1600, txt_DbVar_C1_NvParametersC1_MaxPvgRotTurretCtClkwseRadioPost_0 := 1601, txt_DbVarArrDescr_C1_NvParametersC1_RotTurretCtClkwiseRampRatioTuret := 1602, txt_DbVar_C1_NvParametersC1_RotTurretCtClkwiseRampRatioTuret_0 := 1603, txt_DbVar_C1_NvParametersC1_RotTurretCtClkwiseRampRatioTuret_1 := 1604, txt_DbVarArrDescr_C1_NvParametersC1_RotTurretCtClkwiseRampRatioNacel := 1605, txt_DbVar_C1_NvParametersC1_RotTurretCtClkwiseRampRatioNacel_0 := 1606, txt_DbVar_C1_NvParametersC1_RotTurretCtClkwiseRampRatioNacel_1 := 1607, txt_DbVarArrDescr_C1_NvParametersC1_RotTurretCtClkwiseRampRatioRadio := 1608, txt_DbVar_C1_NvParametersC1_RotTurretCtClkwiseRampRatioRadio_0 := 1609, txt_DbVar_C1_NvParametersC1_RotTurretCtClkwiseRampRatioRadio_1 := 1610, txt_DbVar_C1_NvParametersC1_MinPvgUpAxleOscillant_0 := 1611, txt_DbVar_C1_NvParametersC1_MaxPvgUpAxleOscillant_0 := 1612, txt_DbVarArrDescr_C1_NvParametersC1_PvgUpAxleOscillantRampRatio := 1613, txt_DbVar_C1_NvParametersC1_PvgUpAxleOscillantRampRatio_0 := 1614, txt_DbVar_C1_NvParametersC1_PvgUpAxleOscillantRampRatio_1 := 1615, txt_DbVar_C1_NvParametersC1_MinPvgDownAxleOscillant_0 := 1616, txt_DbVar_C1_NvParametersC1_MaxPvgDownAxleOscillant_0 := 1617, txt_DbVarArrDescr_C1_NvParametersC1_PvgDownAxleOscillantRampRatio := 1618, txt_DbVar_C1_NvParametersC1_PvgDownAxleOscillantRampRatio_0 := 1619, txt_DbVar_C1_NvParametersC1_PvgDownAxleOscillantRampRatio_1 := 1620, txt_DbVar_C1_NvParametersC1_MinPvgUpAxleFixe_0 := 1621, txt_DbVar_C1_NvParametersC1_MaxPvgUpAxleFixe_0 := 1622, txt_DbVarArrDescr_C1_NvParametersC1_PvgUpAxleFixeRampRatio := 1623, txt_DbVar_C1_NvParametersC1_PvgUpAxleFixeRampRatio_0 := 1624, txt_DbVar_C1_NvParametersC1_PvgUpAxleFixeRampRatio_1 := 1625, txt_DbVar_C1_NvParametersC1_MinPvgDownAxleFixe_0 := 1626, txt_DbVar_C1_NvParametersC1_MaxPvgDownAxleFixe_0 := 1627, txt_DbVarArrDescr_C1_NvParametersC1_PvgDownAxleFixeRampRatio := 1628, txt_DbVar_C1_NvParametersC1_PvgDownAxleFixeRampRatio_0 := 1629, txt_DbVar_C1_NvParametersC1_PvgDownAxleFixeRampRatio_1 := 1630, txt_DbVar_C1_NvParametersC1_MinPvgRotFrameCtClkwise_0 := 1631, txt_DbVar_C1_NvParametersC1_MaxPvgRotFrameCtClkwise_0 := 1632, txt_DbVarArrDescr_C1_NvParametersC1_RotFrameCtClkwiseRampRatio := 1633, txt_DbVar_C1_NvParametersC1_RotFrameCtClkwiseRampRatio_0 := 1634, txt_DbVar_C1_NvParametersC1_RotFrameCtClkwiseRampRatio_1 := 1635, txt_DbVar_C1_NvParametersC1_MinPvgRotFrameClkwise_0 := 1636, txt_DbVar_C1_NvParametersC1_MaxPvgRotFrameClkwise_0 := 1637, txt_DbVarArrDescr_C1_NvParametersC1_RotFrameClkwiseRampRatio := 1638, txt_DbVar_C1_NvParametersC1_RotFrameClkwiseRampRatio_0 := 1639, txt_DbVar_C1_NvParametersC1_RotFrameClkwiseRampRatio_1 := 1640, txt_DbVar_C1_NvParametersC1_AntiDemarrageTime_0 := 1641, txt_DbVar_C1_NvParametersC1_TresholdRmpMotorAntidemarrage_0 := 1642, txt_DbVar_C1_NvParametersC1_SlowSpeedUpDeltaArmTelescOut_0 := 1643, txt_DbVar_C1_NvParametersC1_SlowSpeedDownDeltaArmTelescOut_0 := 1644, txt_DbVar_C1_NvParametersC1_SlowSpeedUpArrowArmTelescOut_0 := 1645, txt_DbVar_C1_NvParametersC1_SlowSpeedDownArrowArmTelescOut_0 := 1646, txt_DbVar_C1_NvParametersC1_RotTurretClockSlowSpeedRedAlo_0 := 1647, txt_DbVar_C1_NvParametersC1_RotTurretCtClockSlowSpeedRedAlo_0 := 1648, txt_DbVar_C1_NvParametersC1_ArrowArmDownSlowSpeedRedAlo_0 := 1649, txt_DbVar_C1_NvParametersC1_SlowSpeedRotTurretCtClokTelecOut_0 := 1650, txt_DbVar_C1_NvParametersC1_SlowSpeedRotTurretClokTelecOut_0 := 1651, txt_DbVar_C1_NvParametersC1_MinPvgUpMastMeasure_0 := 1652, txt_DbVar_C1_NvParametersC1_MaxPvgUpMastMeasure_0 := 1653, txt_DbVarArrDescr_C1_NvParametersC1_UpMastMeasureRampRatio := 1654, txt_DbVar_C1_NvParametersC1_UpMastMeasureRampRatio_0 := 1655, txt_DbVar_C1_NvParametersC1_UpMastMeasureRampRatio_1 := 1656, txt_DbVar_C1_NvParametersC1_MinPvgDownMastMeasure_0 := 1657, txt_DbVar_C1_NvParametersC1_MaxPvgDownMastMeasure_0 := 1658, txt_DbVarArrDescr_C1_NvParametersC1_DownMastMeasureRampRatio := 1659, txt_DbVar_C1_NvParametersC1_DownMastMeasureRampRatio_0 := 1660, txt_DbVar_C1_NvParametersC1_DownMastMeasureRampRatio_1 := 1661, txt_DbVar_C1_NvParametersC1_OutCharPosTransmission1Pressure_0 := 1662, txt_DbVar_C1_NvParametersC1_OutCharNeuTransmission1Pressure_0 := 1663, txt_DbVar_C1_NvParametersC1_OutCharNegTransmission1Pressure_0 := 1664, txt_DbVar_C1_NvParametersC1_InCharPosTransmission1Pressure_0 := 1665, txt_DbVar_C1_NvParametersC1_InCharNeuTransmission1Pressure_0 := 1666, txt_DbVar_C1_NvParametersC1_INCharNegTransmission1Pressure_0 := 1667, txt_DbVar_C1_NvParametersC1_OutCharPosTransmission2Pressure_0 := 1668, txt_DbVar_C1_NvParametersC1_OutCharNeuTransmission2Pressure_0 := 1669, txt_DbVar_C1_NvParametersC1_OutCharNegTransmission2Pressure_0 := 1670, txt_DbVar_C1_NvParametersC1_InCharPosTransmission2Pressure_0 := 1671, txt_DbVar_C1_NvParametersC1_InCharNeuTransmission2Pressure_0 := 1672, txt_DbVar_C1_NvParametersC1_INCharNegTransmission2Pressure_0 := 1673, txt_DbVar_C1_NvParametersC1_OutCharPosBypassPressureSensor_0 := 1674, txt_DbVar_C1_NvParametersC1_OutCharNeuBypassPressureSensor_0 := 1675, txt_DbVar_C1_NvParametersC1_OutCharNegBypassPressureSensor_0 := 1676, txt_DbVar_C1_NvParametersC1_InCharPosBypassPressureSensor_0 := 1677, txt_DbVar_C1_NvParametersC1_InCharNeuBypassPressureSensor_0 := 1678, txt_DbVar_C1_NvParametersC1_InCharNegBypassPressureSensor_0 := 1679, txt_DbVar_C1_NvParametersC1_NvParametersC1_1_0 := 1680, txt_DbVar_C1_NvParametersC1_NvParametersC1_2_0 := 1681, txt_DbVar_C1_NvParametersC1_NvParametersC1_3_0 := 1682, txt_DbVar_C1_NvParametersC1_NvParametersC1_4_0 := 1683, txt_DbVar_C1_NvParametersC1_NvParametersC1_5_0 := 1684, txt_DbVar_C1_NvParametersC1_NvParametersC1_6_0 := 1685, txt_DbVar_C1_NvParametersC1_NvParametersC1_7_0 := 1686, txt_DbVar_C1_NvParametersC1_NvParametersC1_8_0 := 1687, txt_DbVar_C1_NvParametersC1_NvParametersC1_9_0 := 1688, txt_DbVar_C1_NvParametersC1_NvParametersC1_10_0 := 1689, txt_DbVar_C1_NvParametersC1_NvParametersC1_11_0 := 1690, txt_DbVar_C1_NvParametersC1_NvParametersC1_12_0 := 1691, txt_DbVar_C1_NvParametersC1_NvParametersC1_13_0 := 1692, txt_DbVar_C1_NvParametersC1_NvParametersC1_14_0 := 1693, txt_DbVar_C1_NvParametersC1_NvParametersC1_15_0 := 1694, txt_DbVar_C1_NvParametersC1_NvParametersC1_16_0 := 1695, txt_DbVar_C1_NvParametersC1_NvParametersC1_17_0 := 1696, txt_DbVar_C1_NvParametersC1_CurFor220VGeneratorOn_0 := 1697, txt_DbVar_C1_NvParametersC1_NbElementTransissionPressure_0 := 1698, txt_DbVar_C1_NvParametersC1_RampUpEvGenerator_0 := 1699, txt_DbVar_C1_NvParametersC1_RampDownEvGenerator_0 := 1700, txt_DbVar_C1_NvParametersC1_GasGaugeAlarm_0 := 1701, txt_DbVar_C1_NvParametersC1_CRC_SRDO1_0 := 1702, txt_DbVar_C1_NvParametersC1_CRC_SRDO2_0 := 1703, txt_DbVar_C1_NvParametersC1_CRC_SRDO3_0 := 1704, txt_DbVar_C1_NvParametersC1_CRC_SRDO4_0 := 1705, txt_DbVar_C1_NvParametersC1_CRC_SRDO5_0 := 1706, txt_DbVar_C1_NvParametersC1_CRC_SRDO6_0 := 1707, txt_DbVar_C1_NvParametersC1_CRC_SRDO7_0 := 1708, txt_DbVar_C1_NvParametersC1_CRC_SRDO8_0 := 1709, txt_DbVar_C1_NvParametersC1_CRC_SRDO9_0 := 1710, txt_DbVar_C1_NvParametersC1_CRC_SRDO10_0 := 1711, txt_DbVar_C1_NvParametersC1_TimeoutSdoRequestTime_0 := 1712, txt_DbVar_C1_NvParametersC1_ActiveSystemFault_0 := 1713, txt_DbVar_C1_NvParametersC1_BypassAlarmActiveC1_0 := 1714, txt_DbVar_C1_NvParametersC1_OutCharPosOilTankTemp_0 := 1715, txt_DbVar_C1_NvParametersC1_OutCharNeuOilTankTemp_0 := 1716, txt_DbVar_C1_NvParametersC1_OutCharNegOilTankTemp_0 := 1717, txt_DbVarArrDescr_C1_NvCalibrationC1_ArmDeltaRampRatioNacellePost := 1718, txt_DbVar_C1_NvCalibrationC1_ArmDeltaRampRatioNacellePost_0 := 1719, txt_DbVar_C1_NvCalibrationC1_ArmDeltaRampRatioNacellePost_1 := 1720, txt_DbVar_C1_NvCalibrationC1_ArmDeltaRampRatioNacellePost_2 := 1721, txt_DbVar_C1_NvCalibrationC1_ArmDeltaRampRatioNacellePost_3 := 1722, txt_DbVarArrDescr_C1_NvCalibrationC1_ArmArrowRampRatioNacellePost := 1723, txt_DbVar_C1_NvCalibrationC1_ArmArrowRampRatioNacellePost_0 := 1724, txt_DbVar_C1_NvCalibrationC1_ArmArrowRampRatioNacellePost_1 := 1725, txt_DbVar_C1_NvCalibrationC1_ArmArrowRampRatioNacellePost_2 := 1726, txt_DbVar_C1_NvCalibrationC1_ArmArrowRampRatioNacellePost_3 := 1727, txt_DbVarArrDescr_C1_NvCalibrationC1_ArmTelescopeRampRatioNacellePost := 1728, txt_DbVar_C1_NvCalibrationC1_ArmTelescopeRampRatioNacellePost_0 := 1729, txt_DbVar_C1_NvCalibrationC1_ArmTelescopeRampRatioNacellePost_1 := 1730, txt_DbVar_C1_NvCalibrationC1_ArmTelescopeRampRatioNacellePost_2 := 1731, txt_DbVar_C1_NvCalibrationC1_ArmTelescopeRampRatioNacellePost_3 := 1732, txt_DbVarArrDescr_C1_NvCalibrationC1_RotTurretRampRatio := 1733, txt_DbVar_C1_NvCalibrationC1_RotTurretRampRatio_0 := 1734, txt_DbVar_C1_NvCalibrationC1_RotTurretRampRatio_1 := 1735, txt_DbVarArrDescr_C1_NvCalibrationC1_PvgEvTorRampRatio := 1736, txt_DbVar_C1_NvCalibrationC1_PvgEvTorRampRatio_0 := 1737, txt_DbVar_C1_NvCalibrationC1_PvgEvTorRampRatio_1 := 1738, txt_DbVar_C1_NvCalibrationC1_PvgEvTorRampRatio_2 := 1739, txt_DbVar_C1_NvCalibrationC1_PvgEvTorRampRatio_3 := 1740, txt_DbVar_C1_NvCalibrationC1_AngleEndStopLowDeltaArm_0 := 1741, txt_DbVar_C1_NvCalibrationC1_AngleCalibEndStopLowDeltaArm_0 := 1742, txt_DbVar_C1_NvCalibrationC1_AngleEndStopHighDeltaArm_0 := 1743, txt_DbVar_C1_NvCalibrationC1_AngleCalibEndStopHighDeltaArm_0 := 1744, txt_DbVar_C1_NvCalibrationC1_AngleEndStopLowArrowArm_0 := 1745, txt_DbVar_C1_NvCalibrationC1_AngleCalibEndStopLowArrowArm_0 := 1746, txt_DbVar_C1_NvCalibrationC1_AngleEndStopHighArrowArm_0 := 1747, txt_DbVar_C1_NvCalibrationC1_AngleCalibEndStopHighArrowArm_0 := 1748, txt_DbVar_C1_NvCalibrationC1_LenghtEndStopLowTelescope1_0 := 1749, txt_DbVar_C1_NvCalibrationC1_LenghtEndStopHighTelescope1_0 := 1750, txt_DbVar_C1_NvCalibrationC1_LenghtCaliEndStopLowTelescope1_0 := 1751, txt_DbVar_C1_NvCalibrationC1_LenghtCaliEndStopHighTelescope1_0 := 1752, txt_DbVar_C1_NvCalibrationC1_LenghtEndStopLowTelescope2_0 := 1753, txt_DbVar_C1_NvCalibrationC1_LenghtEndStopHighTelescope2_0 := 1754, txt_DbVar_C1_NvCalibrationC1_LenghtCaliEndStopLowTelescope2_0 := 1755, txt_DbVar_C1_NvCalibrationC1_LenghtCaliEndStopHighTelescope2_0 := 1756, txt_DbVarArrDescr_C1_NvCalibrationC1_ArmDeltaRampRatioTurretPost := 1757, txt_DbVar_C1_NvCalibrationC1_ArmDeltaRampRatioTurretPost_0 := 1758, txt_DbVar_C1_NvCalibrationC1_ArmDeltaRampRatioTurretPost_1 := 1759, txt_DbVar_C1_NvCalibrationC1_ArmDeltaRampRatioTurretPost_2 := 1760, txt_DbVar_C1_NvCalibrationC1_ArmDeltaRampRatioTurretPost_3 := 1761, txt_DbVarArrDescr_C1_NvCalibrationC1_ArmArrowRampRatioTurretPost := 1762, txt_DbVar_C1_NvCalibrationC1_ArmArrowRampRatioTurretPost_0 := 1763, txt_DbVar_C1_NvCalibrationC1_ArmArrowRampRatioTurretPost_1 := 1764, txt_DbVar_C1_NvCalibrationC1_ArmArrowRampRatioTurretPost_2 := 1765, txt_DbVar_C1_NvCalibrationC1_ArmArrowRampRatioTurretPost_3 := 1766, txt_DbVarArrDescr_C1_NvCalibrationC1_ArmTelescopeRampRatioTurretPost := 1767, txt_DbVar_C1_NvCalibrationC1_ArmTelescopeRampRatioTurretPost_0 := 1768, txt_DbVar_C1_NvCalibrationC1_ArmTelescopeRampRatioTurretPost_1 := 1769, txt_DbVar_C1_NvCalibrationC1_ArmTelescopeRampRatioTurretPost_2 := 1770, txt_DbVar_C1_NvCalibrationC1_ArmTelescopeRampRatioTurretPost_3 := 1771, txt_DbVar_C1_NvCalibrationC1_AngleCalibDeltaArmHyst_0 := 1772, txt_DbVar_C1_NvCalibrationC1_AngleCalibArrowArmHyst_0 := 1773, txt_DbVar_C1_NvCalibrationC1_AngleCalibEndStopHighDeltaArmSla_0 := 1774, txt_DbVar_C1_NvCalibrationC1_AngleCalibEndStopLowDeltaArmSla_0 := 1775, txt_DbVar_C1_NvCalibrationC1_AngleCalibEndStopHighArrowArmSla_0 := 1776, txt_DbVar_C1_NvCalibrationC1_AngleCalibEndStopLowArrowArmSla_0 := 1777, txt_DbVar_C1_Ram48XsInputsC1_UpInclinaisonBasketButton_0 := 1778, txt_DbVar_C1_Ram48XsInputsC1_UpInclinaisonBasketButtonValue_0 := 1779, txt_DbVar_C1_Ram48XsInputsC1_DownInclinaisonBasketButton_0 := 1780, txt_DbVar_C1_Ram48XsInputsC1_DownInclinaisonBasketButtonValue_0 := 1781, txt_DbVar_C1_Ram48XsInputsC1_UpPendularButton_0 := 1782, txt_DbVar_C1_Ram48XsInputsC1_UpPendularButtonValue_0 := 1783, txt_DbVar_C1_Ram48XsInputsC1_DownPendularButton_0 := 1784, txt_DbVar_C1_Ram48XsInputsC1_DownPendularButtonValue_0 := 1785, txt_DbVar_C1_Ram48XsInputsC1_RotationCtClockwiseBasketButton_0 := 1786, txt_DbVar_C1_Ram48XsInputsC1_RotCtClockwiseBasketButtonVal_0 := 1787, txt_DbVar_C1_Ram48XsInputsC1_RotationClockwiseBasketButton_0 := 1788, txt_DbVar_C1_Ram48XsInputsC1_RotationClockwiseBasketButtonVal_0 := 1789, txt_DbVar_C1_Ram48XsInputsC1_Overload1_0 := 1790, txt_DbVar_C1_Ram48XsInputsC1_Overload1Value_0 := 1791, txt_DbVar_C1_Ram48XsInputsC1_Overload2_0 := 1792, txt_DbVar_C1_Ram48XsInputsC1_Overload2Value_0 := 1793, txt_DbVar_C1_Ram48XsInputsC1_NacelleBasketRightSideSensor1_0 := 1794, txt_DbVar_C1_Ram48XsInputsC1_NacelleBasketRightSideSensor1Val_0 := 1795, txt_DbVar_C1_Ram48XsInputsC1_NacelleBasketRightSideSensor2_0 := 1796, txt_DbVar_C1_Ram48XsInputsC1_NacelleBasketRightSideSensor2Val_0 := 1797, txt_DbVar_C1_Ram48XsInputsC1_NacelleBasketLeftSideSensor1_0 := 1798, txt_DbVar_C1_Ram48XsInputsC1_NacelleBasketLeftSideSensor1Val_0 := 1799, txt_DbVar_C1_Ram48XsInputsC1_NacelleBasketLeftSideSensor2_0 := 1800, txt_DbVar_C1_Ram48XsInputsC1_NacelleBasketLeftSideSensor2Val_0 := 1801, txt_DbVar_C1_Ram48XsInputsC1_LowSectorPendularSensor_0 := 1802, txt_DbVar_C1_Ram48XsInputsC1_LowSectorPendularSensorVal_0 := 1803, txt_DbVar_C1_Ram48XsInputsC1_HighSectorPlateSensor_0 := 1804, txt_DbVar_C1_Ram48XsInputsC1_HighSectorPlateSensorVal_0 := 1805, txt_DbVar_C1_Ram48XsInputsC1_FoldedLadderSensor_0 := 1806, txt_DbVar_C1_Ram48XsInputsC1_FoldedLadderSensorVal_0 := 1807, txt_DbVar_C1_Ram48XsInputsC1_SafetyManSystem_0 := 1808, txt_DbVar_C1_Ram48XsInputsC1_DeltaArmAxisJoystick_0 := 1809, txt_DbVar_C1_Ram48XsInputsC1_ArrowArmAxisJoystick_0 := 1810, txt_DbVar_C1_Ram48XsInputsC1_TelescopeArmAxisJoysitck_0 := 1811, txt_DbVar_C1_Ram48XsInputsC1_RotationTurretAxisJoystick_0 := 1812, txt_DbVar_C1_Ram48XsInputsC1_AdvanceAxisJoystick_0 := 1813, txt_DbVar_C1_Ram48XsInputsC1_RearmementSafetyManSystem_0 := 1814, txt_DbVar_C1_Ram48XsInputsC1_RearmementSafetyManSystemVal_0 := 1815, txt_DbVar_C1_Ram48XsInputsC1_AbutementNacelleTrackSide_0 := 1816, txt_DbVar_C1_Ram48XsInputsC1_AbutementNacelleTrackSideVal_0 := 1817, txt_DbVar_C1_Ram48XsInputsC1_AbutementNacelleCenteredSide_0 := 1818, txt_DbVar_C1_Ram48XsInputsC1_AbutementNacelleCenteredSideVal_0 := 1819, txt_DbVar_C1_Ram48XsInputsC1_DeltaArmJystckCenteredTelescope_0 := 1820, txt_DbVar_C1_Ram48XsInputsC1_ArrowJoystickCenteredTurret_0 := 1821, txt_DbVar_C1_Ram48XsInputsC1_CenteredAdvanceJoystick_0 := 1822, txt_DbVar_C1_Ram48XsInputsC1_DeadManPedal_0 := 1823, txt_DbVar_C1_Ram48XsInputsC1_PressenceInNacelleSensor1_0 := 1824, txt_DbVar_C1_Ram48XsInputsC1_PressenceInNacelleSensor2_0 := 1825, txt_DbVar_C1_Ram48XsInputsC1_Gachette_0 := 1826, txt_DbVar_C1_Ram48XsInputsC1_Klaxon_0 := 1827, txt_DbVar_C1_Ram48XsInputsC1_StopMotorButton_0 := 1828, txt_DbVar_C1_Ram48XsInputsC1_AuthorizationWorkKey_0 := 1829, txt_DbVar_C1_Ram48XsInputsC1_EtallonnageJoystickButton_0 := 1830, txt_DbVar_C1_Ram48XsInputsC1_ClosePortillonSensor_0 := 1831, txt_DbVar_C1_Ram48XsInputsC1_Hearbeat48Xs_0 := 1832, txt_DbVar_C1_Ram48XsInputsC1_BatterieVoltage48Xs_0 := 1833, txt_DbVar_C1_RamRcvRadioCmdC1_RotFrameClkwiseButton_0 := 1834, txt_DbVar_C1_RamRcvRadioCmdC1_RotFrameCtClkwiseButton_0 := 1835, txt_DbVar_C1_RamRcvRadioCmdC1_UpPendularOrRotTurretCtClock_0 := 1836, txt_DbVar_C1_RamRcvRadioCmdC1_DownPendularOrRotTurretClock_0 := 1837, txt_DbVar_C1_RamRcvRadioCmdC1_SelectorPendular_0 := 1838, txt_DbVar_C1_RamRcvRadioCmdC1_SelectorRotTurret_0 := 1839, txt_DbVar_C1_RamRcvRadioCmdC1_UpAxleOscillant_0 := 1840, txt_DbVar_C1_RamRcvRadioCmdC1_DownAxleOscillant_0 := 1841, txt_DbVar_C1_RamRcvRadioCmdC1_UpAxleFixe_0 := 1842, txt_DbVar_C1_RamRcvRadioCmdC1_DownAxleFixe_0 := 1843, txt_DbVar_C1_RamRcvRadioCmdC1_ForcingAdvanceTrack_0 := 1844, txt_DbVar_C1_RamLimitMoveC1_AutorizeUpDeltaArm_0 := 1845, txt_DbVar_C1_RamLimitMoveC1_AutorizeDownDeltaArm_0 := 1846, txt_DbVar_C1_RamLimitMoveC1_AutorizeUpArrowArm_0 := 1847, txt_DbVar_C1_RamLimitMoveC1_AutorizeDownArrowArm_0 := 1848, txt_DbVar_C1_RamLimitMoveC1_AutorizeOutTelescopeArm_0 := 1849, txt_DbVar_C1_RamLimitMoveC1_AutorizeInTelescopeArm_0 := 1850, txt_DbVar_C1_RamLimitMoveC1_AutorizeRotBasketClkwise_0 := 1851, txt_DbVar_C1_RamLimitMoveC1_AutorizeRotBasketCtClkwise_0 := 1852, txt_DbVar_C1_RamLimitMoveC1_AutorizeUpInclinaisonBasket_0 := 1853, txt_DbVar_C1_RamLimitMoveC1_AutorizeDownInclinaisonBasket_0 := 1854, txt_DbVar_C1_RamLimitMoveC1_AutorizeUpPendular_0 := 1855, txt_DbVar_C1_RamLimitMoveC1_AutorizeDownPendular_0 := 1856, txt_DbVar_C1_RamLimitMoveC1_AutorizeRotTurretClkwise_0 := 1857, txt_DbVar_C1_RamLimitMoveC1_AutorizeRotTurretCtClkwise_0 := 1858, txt_DbVar_C1_NvParamMotorC1_StartUpCurrentMotor_0 := 1859, txt_DbVar_C1_NvParamMotorC1_HighForcingCurrentMotor_0 := 1860, txt_DbVar_C1_NvParamMotorC1_LowForcingCurrentMotor_0 := 1861, txt_DbVar_C1_NvParamMotorC1_Threshold3_0 := 1862, txt_DbVar_C1_NvParamMotorC1_Threshold2_0 := 1863, txt_DbVar_C1_NvParamMotorC1_Threshold1_0 := 1864, txt_DbVar_C1_NvParamMotorC1_StartUpTime_0 := 1865, txt_DbVar_C1_NvParamMotorC1_HighForcingTime_0 := 1866, txt_DbVar_C1_NvParamMotorC1_TranslationCurrentMotor_0 := 1867, txt_DbVar_C1_NvParamMotorC1_NoMovementCurrentMotor_0 := 1868, txt_DbVar_C1_NvParamMotorC1_TresholdRegimeForGenerator_0 := 1869, txt_DbVar_C1_NvParamMotorC1_EngineIdleSpeedMotor_0 := 1870, txt_DbVar_C1_NvParamMotorC1_CptmaxNoMovement_0 := 1871, txt_DbVar_C1_Ram48XsOutputsC1_MotorDefaultLightErrSta_0 := 1872, txt_DbVar_C1_Ram48XsOutputsC1_MotorDefaultLight_0 := 1873, txt_DbVar_C1_Ram48XsOutputsC1_OverloadLightErrSta_0 := 1874, txt_DbVar_C1_Ram48XsOutputsC1_OverloadLight_0 := 1875, txt_DbVar_C1_Ram48XsOutputsC1_BuzzerErrSta_0 := 1876, txt_DbVar_C1_Ram48XsOutputsC1_Buzzer_0 := 1877, txt_DbVar_C1_Ram48XsOutputsC1_SupplyDeadManPedalAndJoysticks_0 := 1878, txt_DbVar_C1_Ram48XsOutputsC1_WarmingLightErrSta_0 := 1879, txt_DbVar_C1_Ram48XsOutputsC1_WarmingLight_0 := 1880, txt_DbVar_C1_Ram48XsOutputsC1_DeversDefaultLightErrSta_0 := 1881, txt_DbVar_C1_Ram48XsOutputsC1_DeversDefaultLight_0 := 1882, txt_DbVar_C1_Ram48XsOutputsC1_GasOilLightErrSta_0 := 1883, txt_DbVar_C1_Ram48XsOutputsC1_GasOilLight_0 := 1884, txt_DbVar_C1_Ram48XsOutputsC1_WhiteLightARGBasketErrSta_0 := 1885, txt_DbVar_C1_Ram48XsOutputsC1_WhiteLightARGBasket_0 := 1886, txt_DbVar_C1_Ram48XsOutputsC1_RedLightARGBasketErrSta_0 := 1887, txt_DbVar_C1_Ram48XsOutputsC1_RedLightARGBasket_0 := 1888, txt_DbVar_C1_Ram48XsOutputsC1_RedLightARDBasketErrSta_0 := 1889, txt_DbVar_C1_Ram48XsOutputsC1_RedLightARDBasket_0 := 1890, txt_DbVar_C1_Ram48XsOutputsC1_WhiteLightARDBasketErrSta_0 := 1891, txt_DbVar_C1_Ram48XsOutputsC1_WhiteLightARDBasket_0 := 1892, txt_DbVar_C1_Ram48XsOutputsC1_WhiteLightAr15746ErrSta_0 := 1893, txt_DbVar_C1_Ram48XsOutputsC1_WhiteLightAr15746Command_0 := 1894, txt_DbVar_C1_RamEcuC1RcvFromC0_RestrictedModeAruActive_0 := 1895, txt_DbVar_C1_RamEcuC1RcvFromC0_TranslationMovementIsSolicited_0 := 1896, txt_DbVar_C1_RamEcuC1RcvFromC0_AxleMovementIsSolicited_0 := 1897, txt_DbVar_C1_RamEcuC1RcvFromC0_DownAxleFixeSensor_0 := 1898, txt_DbVar_C1_RamEcuC1RcvFromC0_DownAxleOscillantSensor_0 := 1899, txt_DbVar_C1_RamEcuC1RcvFromC0_SlopeAngle_0 := 1900, txt_DbVar_C1_RamEcuC1RcvFromC0_ReduceSpeedRotTurretClockwise_0 := 1901, txt_DbVar_C1_RamEcuC1RcvFromC0_ReduceSpeedRotTurretCounterClock_0 := 1902, txt_DbVar_C1_RamEcuC1RcvFromC0_ReduceSpeedArrowArmDown_0 := 1903, txt_DbVar_C1_RamEcuC1RcvFromC0_StopRotTurretClockwise_0 := 1904, txt_DbVar_C1_RamEcuC1RcvFromC0_StopRotTurretCounterClockwise_0 := 1905, txt_DbVar_C1_RamEcuC1RcvFromC0_StopRotBasketClockwise_0 := 1906, txt_DbVar_C1_RamEcuC1RcvFromC0_StopRotBasketCounterClockwise_0 := 1907, txt_DbVar_C1_RamEcuC1RcvFromC0_StopArrowArmDown_0 := 1908, txt_DbVar_C1_RamEcuC1RcvFromC0_StopTelescopeOut_0 := 1909, txt_DbVar_C1_RamEcuC1RcvFromC0_EncodeurTurret1Angle_0 := 1910, txt_DbVar_C1_RamEcuC1RcvFromC0_RedLightARGBasketCmd_0 := 1911, txt_DbVar_C1_RamEcuC1RcvFromC0_WhiteLightARGBasketCmd_0 := 1912, txt_DbVar_C1_RamEcuC1RcvFromC0_EncodeurMastMeasureRaw_0 := 1913, txt_DbVar_C1_RamEcuC1RcvFromC0_WrongAbutments_0 := 1914, txt_DbVar_C1_RamEcuC1RcvFromC0_SpeedVehicleKmhx100_0 := 1915, txt_DbVar_C1_RamEcuC1RcvFromC0_StopMovementByBrakeTest_0 := 1916, txt_DbVar_C1_RamEcuC1RcvFromC0_StopMovementByBreakInBrake_0 := 1917, txt_DbVar_C1_RamEcuC1RcvFromC0_EnableBuzzerSelectPost_0 := 1918, txt_DbVar_C1_RamEcuC1RcvFromC0_SelectedControlPost_0 := 1919, txt_DbVar_C1_RamEcuC1RcvFromC0_CenteredTurretState_0 := 1920, txt_DbVar_C1_RamEcuC1RcvFromC0_AuthorizeWork_0 := 1921, txt_DbVar_C1_RamEcuC1RcvFromC0_UpOsciAxlePos_0 := 1922, txt_DbVar_C1_RamEcuC1RcvFromC0_UpFixeAxlePos_0 := 1923, txt_DbVar_C1_RamEcuC1RcvFromC0_RailWorkMode_0 := 1924, txt_DbVar_C1_RamEcuC1RcvFromC0_EvForwardCommand_0 := 1925, txt_DbVar_C1_RamEcuC1RcvFromC0_EvBackwardCommand_0 := 1926, txt_DbVar_C1_RamEcuC1RcvFromC0_RedLightARDBasketCmd_0 := 1927, txt_DbVar_C1_RamEcuC1RcvFromC0_WhiteLightARDBasketCmd_0 := 1928, txt_DbVar_C1_RamEcuC1RcvFromC0_SecondParkBrakeActive_0 := 1929, txt_DbVar_C1_RamEcuC1RcvFromC0_AutorisationHighSpeedKeyState_0 := 1930, txt_DbVar_C1_RamEcuC1RcvFromC0_TransRailElectricRampOngoing_0 := 1931, txt_DbVar_C1_RamEcuC1RcvFromC0_RpmPvgTransRail_0 := 1932, txt_DbVar_C1_RamEcuC1RcvFromC0_Batt_Soc_0 := 1933, txt_DbVar_C1_RamEcuC1RcvFromC0_Ibatt_ist_0 := 1934, txt_DbVar_C1_RamEcuC1RcvFromC0_SendAuthorizeReloadBattery_0 := 1935, txt_DbVar_C1_RamEcuEvision7C1_gBattery_On_Off_0 := 1936, txt_DbVar_C1_RamEcuEvision7C1_gPreheat_On_Off_0 := 1937, txt_DbVar_C1_RamEcuEvision7C1_gEngine_Faillure_On_Off_0 := 1938, txt_DbVar_C1_RamEcuEvision7C1_gMaintenance_On_Off_0 := 1939, txt_DbVar_C1_RamEcuEvision7C1_gOil_On_OFF_0 := 1940, txt_DbVar_C1_RamEcuEvision7C1_gDeltaArmSectorDown_0 := 1941, txt_DbVar_C1_RamEcuEvision7C1_gArrowArmSectorDown_0 := 1942, txt_DbVar_C1_RamEcuEvision7C1_gPendularSectorDown_0 := 1943, txt_DbVar_C1_RamEcuEvision7C1_gDeltaArmInCenter_0 := 1944, txt_DbVar_C1_RamEcuEvision7C1_gArrowArmInCenter_0 := 1945, txt_DbVar_C1_RamEcuEvision7C1_gPendularInCenter_0 := 1946, txt_DbVar_C1_RamEcuEvision7C1_gBasketRotationInCenter_0 := 1947, txt_DbVar_C1_RamEcuEvision7C1_gTelescopeInCenter_0 := 1948, txt_DbVar_C1_RamEcuEvision7C1_gBasketInclinaisonInCenter_0 := 1949, txt_DbVar_C1_RamEcuEvision7C1_gDeltaArmMoveUpAllow_0 := 1950, txt_DbVar_C1_RamEcuEvision7C1_gDeltaArmMoveDownAllow_0 := 1951, txt_DbVar_C1_RamEcuEvision7C1_gArrowArmMoveUpAllow_0 := 1952, txt_DbVar_C1_RamEcuEvision7C1_gArrowArmMoveDownAllow_0 := 1953, txt_DbVar_C1_RamEcuEvision7C1_gPendularMoveUpAllow_0 := 1954, txt_DbVar_C1_RamEcuEvision7C1_gPendularMoveDownAllow_0 := 1955, txt_DbVar_C1_RamEcuEvision7C1_gTelescopeMoveOutAllow_0 := 1956, txt_DbVar_C1_RamEcuEvision7C1_gTelescopeMoveInAllow_0 := 1957, txt_DbVar_C1_RamEcuEvision7C1_gTurretCtClockWiseMoveAllow_0 := 1958, txt_DbVar_C1_RamEcuEvision7C1_gTurretClockWiseMoveAllow_0 := 1959, txt_DbVar_C1_RamEcuEvision7C1_gBasketRotCtClockWiseMoveAllow_0 := 1960, txt_DbVar_C1_RamEcuEvision7C1_gBasketRotClockWiseMoveAllow_0 := 1961, txt_DbVar_C1_RamEcuEvision7C1_gBasketInclinaisonMoveUpAllow_0 := 1962, txt_DbVar_C1_RamEcuEvision7C1_gBasketInclinaisonMoveDownAllow_0 := 1963, txt_DbVar_C1_RamEcuEvision7C1_gVehiculeDefault_0 := 1964, txt_DbVar_C1_RamEcuEvision7C1_gTelescopeOutputPossible_0 := 1965, txt_DbVar_C1_RamEcuEvision7C1_gTelescopeWinderFault_0 := 1966, txt_DbVar_C1_RamEcuEvision7C1_gNacellePostSelector_0 := 1967, txt_DbVar_C1_RamEcuEvision7C1_gSTOP_On_Off_0 := 1968, txt_DbVar_C1_RamEcuEvision7C1_gSafeManSystem_0 := 1969, txt_DbVar_C1_RamEcuEvision7C1_gHighSpeedAllow_0 := 1970, txt_DbVar_C1_RamEcuEvision7C1_gAutomatiqueStop_0 := 1971, txt_DbVar_C1_RamEcuEvision7C1_gLowSpeedByFault_0 := 1972, txt_DbVar_C1_RamEcuEvision7C1_gMeasuringMastFault_0 := 1973, txt_DbVar_C1_RamEcuEvision7C1_gFuel_0 := 1974, txt_DbVar_C1_RamEcuEvision7C1_gBattery_Voltage_0 := 1975, txt_DbVar_C1_RamEcuEvision7C1_gTrainTransmissionPressure_0 := 1976, txt_DbVar_C1_RamEvision4C1_LifeByte_0 := 1977, txt_DbVar_C1_RamEvision4C1_gDelta_Arm_Move_Up_0 := 1978, txt_DbVar_C1_RamEvision4C1_gDelta_Arm_Move_Down_0 := 1979, txt_DbVar_C1_RamEvision4C1_gArrow_Move_Up_0 := 1980, txt_DbVar_C1_RamEvision4C1_gArrow_Move_Down_0 := 1981, txt_DbVar_C1_RamEvision4C1_gPendular_Move_Up_0 := 1982, txt_DbVar_C1_RamEvision4C1_gPendular_Move_Down_0 := 1983, txt_DbVar_C1_RamEvision4C1_gTelescope_Move_Out_0 := 1984, txt_DbVar_C1_RamEvision4C1_gTelescope_Move_In_0 := 1985, txt_DbVar_C1_RamEvision4C1_gBasket_Inclinaison_Move_Up_0 := 1986, txt_DbVar_C1_RamEvision4C1_gBasket_Inclinaison_Move_Down_0 := 1987, txt_DbVar_C1_RamEvision4C1_gTurret_Rotate_ClockWise_0 := 1988, txt_DbVar_C1_RamEvision4C1_gTurret_Rotate_Counter_ClockWise_0 := 1989, txt_DbVar_C1_RamEvision4C1_gBasket_Rotate_ClockWise_0 := 1990, txt_DbVar_C1_RamEvision4C1_gBasket_Rotate_Counter_ClockWise_0 := 1991, txt_DbVar_C1_RamEvision4C1_gKeyRpmSelect_0 := 1992, txt_DbVar_C1_RamEvision4C1_gKeyRpmOff_0 := 1993, txt_DbVar_C1_RamEvision4C1_gForcingWhiteRaillight_0 := 1994, txt_DbVar_C1_RamEvision4C1_gForcingNeons_0 := 1995, txt_DbVar_C1_RamEvision4C1_gKeyCalibMin_0 := 1996, txt_DbVar_C1_RamEvision4C1_gKeyCalibMax_0 := 1997, txt_DbVar_C1_RamEvision4C1_gKeyCalibValid_0 := 1998, txt_DbVar_C1_RamEvision4C1_gElementChoice_0 := 1999, txt_DbVar_C1_RamEvision4C1_gKeyCalibMax2_0 := 2000, txt_DbVar_C1_RamEvision4C1_gKeySlopeLgReset_0 := 2001, txt_DbVar_C1_RamEvision4C1_gKeySlopeTrReset_0 := 2002, txt_DbVar_C1_RamEvision4C1_ActivePageOpus_0 := 2003, txt_DbVar_C1_RamEvision4C1_KeyYesReloadWithGenerator_0 := 2004, txt_DbVar_C1_RamEvision4C1_KeyNoReloadWithGenerator_0 := 2005, txt_DbVar_C1_RamEcuCaliCmdC1_CalibAngleEndStopLowDeltaArm_0 := 2006, txt_DbVar_C1_RamEcuCaliCmdC1_CalibAngleEndStopHighDeltaArm_0 := 2007, txt_DbVar_C1_RamEcuCaliCmdC1_CalibAngleEndStopLowArrowArm_0 := 2008, txt_DbVar_C1_RamEcuCaliCmdC1_CalibAngleEndStopHighArrowArm_0 := 2009, txt_DbVar_C1_RamEcuCaliCmdC1_SavedCalibrationListC1_0 := 2010, txt_DbVar_C1_RamEcuCaliCmdC1_CalibLenghtEndStopLowTelescope_0 := 2011, txt_DbVar_C1_RamEcuCaliCmdC1_CalibLenghtEndStopHighTelescope_0 := 2012, txt_DbVarArrDescr_C1_NvParamLimitWorkEnvelopeC1_SlopeTelescModeCurveSlopeAngles := 2013, txt_DbVar_C1_NvParamLimitWorkEnvelopeC1_SlopeTelescModeCurveSlopeAngles_0 := 2014, txt_DbVar_C1_NvParamLimitWorkEnvelopeC1_SlopeTelescModeCurveSlopeAngles_1 := 2015, txt_DbVar_C1_NvParamLimitWorkEnvelopeC1_SlopeTelescModeCurveSlopeAngles_2 := 2016, txt_DbVar_C1_NvParamLimitWorkEnvelopeC1_SlopeTelescModeCurveSlopeAngles_3 := 2017, txt_DbVar_C1_NvParamLimitWorkEnvelopeC1_SlopeTelescModeCurveSlopeAngles_4 := 2018, txt_DbVar_C1_NvParamLimitWorkEnvelopeC1_SlopeTelescModeCurveSlopeAngles_5 := 2019, txt_DbVar_C1_NvParamLimitWorkEnvelopeC1_SlopeTelescModeCurveSlopeAngles_6 := 2020, txt_DbVar_C1_NvParamLimitWorkEnvelopeC1_SlopeTelescModeCurveSlopeAngles_7 := 2021, txt_DbVar_C1_NvParamLimitWorkEnvelopeC1_SlopeTelescModeCurveSlopeAngles_8 := 2022, txt_DbVarArrDescr_C1_NvParamLimitWorkEnvelopeC1_SlopeTelescModeCurveTelescLenght := 2023, txt_DbVar_C1_NvParamLimitWorkEnvelopeC1_SlopeTelescModeCurveTelescLenght_0 := 2024, txt_DbVar_C1_NvParamLimitWorkEnvelopeC1_SlopeTelescModeCurveTelescLenght_1 := 2025, txt_DbVar_C1_NvParamLimitWorkEnvelopeC1_SlopeTelescModeCurveTelescLenght_2 := 2026, txt_DbVar_C1_NvParamLimitWorkEnvelopeC1_SlopeTelescModeCurveTelescLenght_3 := 2027, txt_DbVar_C1_NvParamLimitWorkEnvelopeC1_SlopeTelescModeCurveTelescLenght_4 := 2028, txt_DbVar_C1_NvParamLimitWorkEnvelopeC1_SlopeTelescModeCurveTelescLenght_5 := 2029, txt_DbVar_C1_NvParamLimitWorkEnvelopeC1_SlopeTelescModeCurveTelescLenght_6 := 2030, txt_DbVar_C1_NvParamLimitWorkEnvelopeC1_SlopeTelescModeCurveTelescLenght_7 := 2031, txt_DbVar_C1_NvParamLimitWorkEnvelopeC1_SlopeTelescModeCurveTelescLenght_8 := 2032, txt_DbVar_C1_NvParamLimitWorkEnvelopeC1_TelescopeLimitCriticZoneThresRel_0 := 2033, txt_DbVar_C1_NvParamLimitWorkEnvelopeC1_TelescopeLimitCriticZoneHystRel_0 := 2034, txt_DbVar_C1_NvParamLimitWorkEnvelopeC1_DeltaArmLimitSlopeHighThresAbs_0 := 2035, txt_DbVar_C1_NvParamLimitWorkEnvelopeC1_DeltaArmLimitSlopeHighHystRel_0 := 2036, txt_DbVar_C1_NvParamLimitWorkEnvelopeC1_DeltaArmLimitUpperZoneThresAbs_0 := 2037, txt_DbVar_C1_NvParamLimitWorkEnvelopeC1_DeltaArmLimitUpperZoneHystRel_0 := 2038, txt_DbVar_C1_NvParamLimitWorkEnvelopeC1_DeltaArmLimitSlowZoneThresRel_0 := 2039, txt_DbVar_C1_NvParamLimitWorkEnvelopeC1_DeltaArmLimitSlowSpeedReduc_0 := 2040, txt_DbVar_C1_NvParamLimitWorkEnvelopeC1_DeltaArmLimitCriticZoneThresRel_0 := 2041, txt_DbVar_C1_NvParamLimitWorkEnvelopeC1_DeltaArmLimitCriticZoneHystRel_0 := 2042, txt_DbVar_C1_NvParamLimitWorkEnvelopeC1_ArrowArmLimitLowerZoneThresAbs_0 := 2043, txt_DbVar_C1_NvParamLimitWorkEnvelopeC1_ArrowArmLimitLowerZoneHystRel_0 := 2044, txt_DbVar_C1_NvParamLimitWorkEnvelopeC1_ArrowArmLimitSlowZoneThresRel_0 := 2045, txt_DbVar_C1_NvParamLimitWorkEnvelopeC1_ArrowArmLimitSlowSpeedReduc_0 := 2046, txt_DbVar_C1_NvParamLimitWorkEnvelopeC1_ArrowArmLimitCriticZoneThresRel_0 := 2047, txt_DbVar_C1_NvParamLimitWorkEnvelopeC1_ArrowArmLimitCriticZoneHystRel_0 := 2048, txt_DbVarArrDescr_C1_NvParamLimitWorkEnvelopeC1_ArmTelescModeCurveArmAngles := 2049, txt_DbVar_C1_NvParamLimitWorkEnvelopeC1_ArmTelescModeCurveArmAngles_0 := 2050, txt_DbVar_C1_NvParamLimitWorkEnvelopeC1_ArmTelescModeCurveArmAngles_1 := 2051, txt_DbVar_C1_NvParamLimitWorkEnvelopeC1_ArmTelescModeCurveArmAngles_2 := 2052, txt_DbVar_C1_NvParamLimitWorkEnvelopeC1_ArmTelescModeCurveArmAngles_3 := 2053, txt_DbVar_C1_NvParamLimitWorkEnvelopeC1_ArmTelescModeCurveArmAngles_4 := 2054, txt_DbVar_C1_NvParamLimitWorkEnvelopeC1_ArmTelescModeCurveArmAngles_5 := 2055, txt_DbVar_C1_NvParamLimitWorkEnvelopeC1_ArmTelescModeCurveArmAngles_6 := 2056, txt_DbVar_C1_NvParamLimitWorkEnvelopeC1_ArmTelescModeCurveArmAngles_7 := 2057, txt_DbVar_C1_NvParamLimitWorkEnvelopeC1_ArmTelescModeCurveArmAngles_8 := 2058, txt_DbVarArrDescr_C1_NvParamLimitWorkEnvelopeC1_ArmTelescModeCurveTelescLenght := 2059, txt_DbVar_C1_NvParamLimitWorkEnvelopeC1_ArmTelescModeCurveTelescLenght_0 := 2060, txt_DbVar_C1_NvParamLimitWorkEnvelopeC1_ArmTelescModeCurveTelescLenght_1 := 2061, txt_DbVar_C1_NvParamLimitWorkEnvelopeC1_ArmTelescModeCurveTelescLenght_2 := 2062, txt_DbVar_C1_NvParamLimitWorkEnvelopeC1_ArmTelescModeCurveTelescLenght_3 := 2063, txt_DbVar_C1_NvParamLimitWorkEnvelopeC1_ArmTelescModeCurveTelescLenght_4 := 2064, txt_DbVar_C1_NvParamLimitWorkEnvelopeC1_ArmTelescModeCurveTelescLenght_5 := 2065, txt_DbVar_C1_NvParamLimitWorkEnvelopeC1_ArmTelescModeCurveTelescLenght_6 := 2066, txt_DbVar_C1_NvParamLimitWorkEnvelopeC1_ArmTelescModeCurveTelescLenght_7 := 2067, txt_DbVar_C1_NvParamLimitWorkEnvelopeC1_ArmTelescModeCurveTelescLenght_8 := 2068, txt_DbVar_C1_NvParamLimitWorkEnvelopeC1_SlopeTelescopeMode_0 := 2069, txt_DbVar_C1_NvParamLimitWorkEnvelopeC1_ArrowArmPerformLowUpperSector_0 := 2070, txt_DbVar_C1_NvParamLimitWorkEnvelopeC1_ArrowArmPerformSectorUpperCritic_0 := 2071, txt_DbVar_C1_NvParamLimitWorkEnvelopeC1_ArrowArmPerformSectorHyst_0 := 2072, txt_DbVar_C1_RamLimitWorkEnvelopeC1_ReduceSpeedDeltaArmUp_0 := 2073, txt_DbVar_C1_RamLimitWorkEnvelopeC1_ReduceSpeedArrowArmDown_0 := 2074, txt_DbVar_C1_RamLimitWorkEnvelopeC1_StopTelescopeOut_0 := 2075, txt_DbVar_C1_RamLimitWorkEnvelopeC1_StopDeltaArmUp_0 := 2076, txt_DbVar_C1_RamLimitWorkEnvelopeC1_StopArrowArmDown_0 := 2077, txt_DbVar_C1_RamLimitWorkEnvelopeC1_StopAllMovements_0 := 2078, txt_DbVar_C1_RamLimitWorkEnvelopeC1_SelectedSlopeAngle_0 := 2079, txt_DbVar_C1_RamLimitWorkEnvelopeC1_TelescopeLimitStrokeThres_0 := 2080, txt_DbVar_C1_RamLimitWorkEnvelopeC1_TelescopeInCriticalZone_0 := 2081, txt_DbVar_C1_RamLimitWorkEnvelopeC1_SlopeIsHigh_0 := 2082, txt_DbVar_C1_RamLimitWorkEnvelopeC1_DeltaArmInUpperZone_0 := 2083, txt_DbVar_C1_RamLimitWorkEnvelopeC1_DeltaArmInCriticalZone_0 := 2084, txt_DbVar_C1_RamLimitWorkEnvelopeC1_ArrowArmInLowerZone_0 := 2085, txt_DbVar_C1_RamLimitWorkEnvelopeC1_ArrowArmInCriticalZone_0 := 2086, txt_DbVar_C1_RamLimitWorkEnvelopeC1_EnableSimuMode_0 := 2087, txt_DbVar_C1_RamLimitWorkEnvelopeC1_SimuSlopeAngleLong_0 := 2088, txt_DbVar_C1_RamLimitWorkEnvelopeC1_SimuSlopeAngleTrans_0 := 2089, txt_DbVar_C1_RamLimitWorkEnvelopeC1_SimuTelescopePositionSensor_0 := 2090, txt_DbVar_C1_RamLimitWorkEnvelopeC1_SimuDeltaArmAngularSensor_0 := 2091, txt_DbVar_C1_RamLimitWorkEnvelopeC1_SimuArrowArmAngularSensor_0 := 2092, txt_DbVar_C1_RamTelescopeCanC1_StateHeartBeatTelescopeSensor_0 := 2093, txt_DbVar_C1_RamTelescopeCanC1_LenghtTelescope1_0 := 2094, txt_DbVar_C1_RamTelescopeCanC1_ErrorRetractorTelescope1_0 := 2095, txt_DbVar_C1_RamTelescopeCanC1_RetractorTelescopeVal1_0 := 2096, txt_DbVar_C1_RamTelescopeCanC1_LenghtTelescope2_0 := 2097, txt_DbVar_C1_RamTelescopeCanC1_ErrorRetractorTelescope2_0 := 2098, txt_DbVar_C1_RamTelescopeCanC1_RetractorTelescopeVal2_0 := 2099, txt_DbVar_C1_RamMvtEndStopC1_ReduceSpeedRotTurretClockwise_0 := 2100, txt_DbVar_C1_RamMvtEndStopC1_StopRotTurretClockwise_0 := 2101, txt_DbVar_C1_RamMvtEndStopC1_ReduceSpeedRotTurretCounterClock_0 := 2102, txt_DbVar_C1_RamMvtEndStopC1_StopRotTurretCounterClockwise_0 := 2103, txt_DbVar_C1_RamMvtEndStopC1_ReduceSpeedDeltaArmDown_0 := 2104, txt_DbVar_C1_RamMvtEndStopC1_FoldedDeltaArm_0 := 2105, txt_DbVar_C1_RamMvtEndStopC1_ReduceSpeedDeltaArmUp_0 := 2106, txt_DbVar_C1_RamMvtEndStopC1_TestTurretPosition_0 := 2107, txt_DbVar_C1_RamMvtEndStopC1_TestDeltaArmPosition_0 := 2108, txt_DbVar_C1_RamMvtEndStopC1_FoldedArrowArm_0 := 2109, txt_DbVar_C1_RamMvtEndStopC1_ReduceSpeedArrowArmUp_0 := 2110, txt_DbVar_C1_RamMvtEndStopC1_ReduceSpeedArrowArmDown_0 := 2111, txt_DbVar_C1_RamMvtEndStopC1_ReduceSpeedTelescopFolded_0 := 2112, txt_DbVar_C1_RamMvtEndStopC1_ReduceSpeedTelescopeUp_0 := 2113, txt_DbVar_C1_RamMvtEndStopC1_ReduceSpeedTelescopeDown_0 := 2114, txt_DbVar_C1_RamMvtEndStopC1_PerformFoldedTelescopeStop_0 := 2115, txt_DbVar_C1_RamMvtEndStopC1_PerformAutoriseTransSlopeArrow_0 := 2116, txt_DbVar_C1_RamMvtEndStopC1_ValidSectorTelescope_0 := 2117, txt_DbVar_C1_RamMvtEndStopC1_ValidFirstSectorTelescope_0 := 2118, txt_DbVar_C1_NvParamMvtEndStopC1_TurretNegEndStopThres_0 := 2119, txt_DbVar_C1_NvParamMvtEndStopC1_TurretNegEndStopHyst_0 := 2120, txt_DbVar_C1_NvParamMvtEndStopC1_TurretNegEndStopSlowThres_0 := 2121, txt_DbVar_C1_NvParamMvtEndStopC1_TurretPosEndStopThres_0 := 2122, txt_DbVar_C1_NvParamMvtEndStopC1_TurretPosEndStopHyst_0 := 2123, txt_DbVar_C1_NvParamMvtEndStopC1_TurretPosEndStopSlowThres_0 := 2124, txt_DbVar_C1_NvParamMvtEndStopC1_FoldedDeltaArmThres_0 := 2125, txt_DbVar_C1_NvParamMvtEndStopC1_FoldedDeltaArmHyst_0 := 2126, txt_DbVar_C1_NvParamMvtEndStopC1_DeltaArmBottomEndStopSlowThres_0 := 2127, txt_DbVar_C1_NvParamMvtEndStopC1_DeltaArmTopEndStopThres_0 := 2128, txt_DbVar_C1_NvParamMvtEndStopC1_DeltaArmTopEndStopHyst_0 := 2129, txt_DbVar_C1_NvParamMvtEndStopC1_DeltaArmTopEndStopSlowThres_0 := 2130, txt_DbVar_C1_NvParamMvtEndStopC1_FoldedArrowArmThres_0 := 2131, txt_DbVar_C1_NvParamMvtEndStopC1_FoldedArrowArmHyst_0 := 2132, txt_DbVar_C1_NvParamMvtEndStopC1_DeltaArmSlowMvtEndStop_0 := 2133, txt_DbVar_C1_NvParamMvtEndStopC1_ArrowArmTopEndStopSlowThres_0 := 2134, txt_DbVar_C1_NvParamMvtEndStopC1_ArrowArmBottomEndStopSlowThres_0 := 2135, txt_DbVar_C1_NvParamMvtEndStopC1_ArrowArmTopEndStopThres_0 := 2136, txt_DbVar_C1_NvParamMvtEndStopC1_ArrowArmSlowMvtDownEndStop_0 := 2137, txt_DbVar_C1_NvParamMvtEndStopC1_ArrowArmSlowMvtUpEndStop_0 := 2138, txt_DbVar_C1_NvParamMvtEndStopC1_TelescopSlowMvtFoldedEndStop_0 := 2139, txt_DbVar_C1_NvParamMvtEndStopC1_TelescopePerfOutLimit_0 := 2140, txt_DbVar_C1_NvParamMvtEndStopC1_TelescopePerfOutLimitHyst_0 := 2141, txt_DbVar_C1_NvParamMvtEndStopC1_TelescopePerfOutLimitSlowThres_0 := 2142, txt_DbVar_C1_NvParamAutoStopC1_TurretRearCenterPos_0 := 2143, txt_DbVar_C1_NvParamAutoStopC1_TurretFrontPositiveCenterPos_0 := 2144, txt_DbVar_C1_NvParamAutoStopC1_TurretFrontNegativeCenterPos_0 := 2145, txt_DbVar_C1_NvParamAutoStopC1_TurretCenterZoneWindow_0 := 2146, txt_DbVar_C1_NvParamAutoStopC1_TurretCenterZoneWindowHyst_0 := 2147, txt_DbVar_C1_NvParamAutoStopC1_TurretCenterZoneSlowThres_0 := 2148, txt_DbVar_C1_NvParamAutoStopC1_TurretCenterZoneWindowLeft_0 := 2149, txt_DbVar_C1_NvParamAutoStopC1_TurretCenterZoneWindowRight_0 := 2150, txt_DbVar_C1_RamAutoStopC1_StopBasketRotation_0 := 2151, txt_DbVar_C1_RamAutoStopC1_StopTurretRotation_0 := 2152, txt_DbVar_C1_RamAutoStopC1_ReduceSpeedRotTurretClockwise_0 := 2153, txt_DbVar_C1_RamAutoStopC1_ReduceSpeedRotTurretCounterClock_0 := 2154, txt_DbVar_C1_RamAutoStopC1_TurrentInCenterPos_0 := 2155, txt_DbVar_C1_RamAutoStopC1_EnableSimuMode_0 := 2156, txt_DbVar_C1_RamAutoStopC1_TestBasketLeftSideSensor_0 := 2157, txt_DbVar_C1_RamAutoStopC1_TestBasketRightSideSensor_0 := 2158, txt_DbVar_C1_RamAutoStopC1_TestBasketRotCmdEnabled_0 := 2159, txt_DbVar_C1_RamAutoStopC1_TestTurretAngularPosition_0 := 2160, txt_DbVar_C1_RamAutoStopC1_TestTurretRotCmdEnabled_0 := 2161, txt_DbVar_C1_RamAutoStopC1_TurretInRearCenterPos_0 := 2162, txt_DbVar_C1_RamAutoStopC1_TurretInFrontPositiveCenterPos_0 := 2163, txt_DbVar_C1_RamAutoStopC1_TurretInFrontNegativeCenterPos_0 := 2164, txt_DbVar_C1_RamAutoStopC1_BasketInCentrerPos_0 := 2165, txt_DbVar_C1_RamAutoStopC1_TurretRotationCmdEnabled_0 := 2166, txt_DbVar_C1_RamAutoStopC1_CounterStopTurretRotationDebug_0 := 2167, txt_DbVar_C1_RamAutoStopC1_CounterNoStopTurretRotationDebug_0 := 2168, txt_DbVar_C1_RamMastMeasureC1_Fonction_Active_0 := 2169, txt_DbVar_C1_RamMastMeasureC1_Commande_Neutre_0 := 2170, txt_DbVar_C1_RamMastMeasureC1_Authorize_Driving_0 := 2171, txt_DbVar_C1_RamMastMeasureC1_Folded_Position_Mast_0 := 2172, txt_DbVar_C1_RamMastMeasureC1_Stop_Movement_By_Mast_0 := 2173, txt_DbVar_C1_RamMastMeasureC1_RazDistanceTraveledButton_0 := 2174, txt_DbVar_C1_RamMastMeasureC1_DistanceTraveledMm_0 := 2175, txt_DbVar_C1_RamMastMeasureC1_DeltaMinMaxEncodeurValue_0 := 2176, txt_DbVar_C1_RamMastMeasureC1_EncodeurMastCentimeterOffset_0 := 2177, txt_DbVar_C1_RamMastMeasureC1_EncodeurMastMeasureCentimeter_0 := 2178, txt_DbVar_C1_RamMastMeasureC1_NoMovementIsDuringAndNeutralCmd_0 := 2179, txt_DbVar_C1_RamMastMeasureC1_ScalingJoyMatTelescope_0 := 2180, txt_DbVar_C1_RamMastMeasureC1_TimeWithMastNotFolded_0 := 2181, txt_DbVar_C1_RamMastMeasureC1_DownAxleOscillantForMast_0 := 2182, txt_DbVar_C1_RamMastMeasureC1_VisibleDistanceTraveledMat_0 := 2183, txt_DbVar_C1_RamMastMeasureC1_MastInUpperPosition_0 := 2184, txt_DbVar_C1_RamMastMeasureC1_MastPanthoInFoldedPosition_0 := 2185, txt_DbVar_C1_RamMastMeasureC1_ValveInDownPosition_0 := 2186, txt_DbVar_C1_RamMastMeasureC1_PostInterdictionMastSNCF_0 := 2187, txt_DbVar_C1_RamMastMeasureC1_MemoFirstValidCycleMast_0 := 2188, txt_DbVar_C1_RamMastMeasureC1_ContactMastAutorisationOfMvts_0 := 2189, txt_DbVar_C1_RamMastMeasureC1_InterdictionOfNacelleTurretPost_0 := 2190, txt_DbVar_C1_RamMastMeasureC1_PictoWarningFirstValidCycleMast_0 := 2191, txt_DbVar_C1_NvParamMastC1_Offset_Mast_Centimeter_0 := 2192, txt_DbVar_C1_NvParamMastC1_FoldedMastThres_0 := 2193, txt_DbVar_C1_NvParamMastC1_FoldedMastHyst_0 := 2194, txt_DbVar_C1_NvParamMastC1_MinValueEncodeurMast_0 := 2195, txt_DbVar_C1_NvParamMastC1_MaxValueEncodeurMast_0 := 2196, txt_DbVar_C1_NvParamMastC1_MinCentimeterEncodeurMast_0 := 2197, txt_DbVar_C1_NvParamMastC1_MaxCentimeterEncodeurMast_0 := 2198, txt_DbVar_C1_NvParamMastC1_MastDisplayRefreshCycleTime_0 := 2199, txt_DbVar_C1_RamEvision7C1_gActivateMeasuringMast_0 := 2200, txt_DbVar_C1_RamEvision7C1_gButtonCalibMinMastMeasure_0 := 2201, txt_DbVar_C1_RamEvision7C1_gButtonCalibMaxMastMeasure_0 := 2202, txt_DbVar_C1_RamEvision7C1_SavePosEncodeurMastMeasureButton_0 := 2203, txt_DbVar_C1_RamEvision7C1_RazDistanceTraveledMastMeasure_0 := 2204, txt_DbVar_C1_RamEvision7C1_gSerialNumber_0 := 2205, txt_DbVar_C1_RamEvision7C1_gBPBasketValidate_0 := 2206, txt_DbVar_C1_RamEvision7C1_gKeyFilterOverload_0 := 2207, txt_DbVar_C1_RamEvision7C1_gKeyNextMode_0 := 2208, txt_DbVar_C1_RamEvision7C1_gKeyPrevMode_0 := 2209, txt_DbVar_C1_RamEvision7C1_gKeySignalDanger_0 := 2210, txt_DbVar_C1_RamEvision7C1_gKeyFlashLightON_0 := 2211, txt_DbVar_C1_RamEvision7C1_gKeyCalibMastMin_0 := 2212, txt_DbVar_C1_RamEvision7C1_gKeyCalibMastMax_0 := 2213, txt_DbVar_C1_RamEvision7C1_gKeyCalibMastValid_0 := 2214, txt_DbVar_C1_RamEvision7C1_gKeyGeneratorActivate_0 := 2215, txt_DbVar_C1_NvParamAlarmC1_BypassPressureThres_0 := 2216, txt_DbVar_C1_NvParamAlarmC1_TelescopeInToleranceInductive_0 := 2217, txt_DbVar_C1_NvParamAlarmC1_TelescopeToleranceNoMovement_0 := 2218, txt_DbVar_C1_NvParamAlarmC1_TelescopeToleranceChannels_0 := 2219, txt_DbVar_C1_NvParamAlarmC1_AlternatorRegimeMaxThres_0 := 2220, txt_DbVar_C1_NvParamAlarmC1_BatteryVoltageMinThres_0 := 2221, txt_DbVar_C1_NvParamAlarmC1_MinAlarmJoyDeltaArmPrctBat_0 := 2222, txt_DbVar_C1_NvParamAlarmC1_MaxAlarmJoyDeltaArmPrctBat_0 := 2223, txt_DbVar_C1_NvParamAlarmC1_MinAlarmJoyArrowArmPrctBat_0 := 2224, txt_DbVar_C1_NvParamAlarmC1_MaxAlarmJoyArrowArmPrctBat_0 := 2225, txt_DbVar_C1_NvParamAlarmC1_MinAlarmJoyTelescopeArmPrctBat_0 := 2226, txt_DbVar_C1_NvParamAlarmC1_MaxAlarmJoyTelescopeArmPrctBat_0 := 2227, txt_DbVar_C1_NvParamAlarmC1_MinAlarmJoyRotTurretArmPrctBat_0 := 2228, txt_DbVar_C1_NvParamAlarmC1_MaxAlarmJoyRotTurretArmPrctBat_0 := 2229, txt_DbVar_C1_NvParamAlarmC1_MinAlarmJoyAdvancementPrctBat_0 := 2230, txt_DbVar_C1_NvParamAlarmC1_MaxAlarmJoyAdvancementPrctBat_0 := 2231, txt_DbVar_C1_NvParamAlarmC1_TimeBypassFault_0 := 2232, txt_DbVar_C1_NvParamAlarmC1_cptTimeTestBypassMax_0 := 2233, txt_DbVar_C1_RamEcuC1RcvFailluresFromC0_Dm_Swi_Dbl_NcNo_Inc_FrameRot_0 := 2234, txt_DbVar_C1_RamEcuC1RcvFailluresFromC0_Dm_Turret_Sensor_Fault_0 := 2235, txt_DbVar_C1_RamEcuC1RcvFailluresFromC0_EvParkBrakeAxleOscillantFault_0 := 2236, txt_DbVar_C1_RamEcuC1RcvFailluresFromC0_EvParkBrakeAxleFixeFault_0 := 2237, txt_DbVar_C1_RamEcuC1RcvFailluresFromC0_EvServiceBrakeAxleOscillantFault_0 := 2238, txt_DbVar_C1_RamEcuC1RcvFailluresFromC0_EvServiceBrakeAxleFixeFault_0 := 2239, txt_DbVar_C1_RamEcuC1RcvFailluresFromC0_EvServiceBrakeTrackFault_0 := 2240, txt_DbVar_C1_RamEcuC1RcvFailluresFromC0_Rm_Com_Can_Radio_Loss_0 := 2241, txt_DbVar_C1_RamEcuC1RcvFailluresFromC0_Ev2ndParkBrakeAxleFixeFault_0 := 2242, txt_DbVar_C1_RamEcuC1RcvFailluresFromC0_Ev2ndParkBrakeAxleOsciFault_0 := 2243, txt_DbVar_C1_RamData4C1RcvFromC0_StopAggravantMovements_0 := 2244, txt_DbVar_C1_RamData4C1RcvFromC0_TurretPostorRadoPostOn_0 := 2245, txt_DbVar_C1_RamData4C1RcvFromC0_MotorAccelerated_0 := 2246, txt_DbVar_C1_RamData4C1RcvFromC0_RadioPostSelectorOn_0 := 2247, txt_DbVar_C1_RamData4C1RcvFromC0_SlopeHighWithWorkOnCrawler_0 := 2248, txt_DbVar_C1_RamData4C1RcvFromC0_ErrorActiveOnC0_0 := 2249, txt_DbVar_C1_RamData4C1RcvFromC0_RailWorkMultiLaneMode_0 := 2250, txt_DbVar_C1_RamData4C1RcvFromC0_TestFrance_0 := 2251, txt_DbVar_C1_RamData4C1RcvFromC0_WhiteLightAV15746Command_0 := 2252, txt_DbVar_C1_RamData4C1RcvFromC0_WhiteLightAr15746Command_0 := 2253, txt_DbVar_C1_RamData4C1RcvFromC0_Signal_9_0 := 2254, txt_DbVar_C1_RamData4C1RcvFromC0_Signal_10_0 := 2255, txt_DbVar_C1_RamData4C1RcvFromC0_Signal_11_0 := 2256, txt_DbVar_C1_RamData4C1RcvFromC0_AddPerformanceFunc_0 := 2257, txt_DbVar_C1_RamData4C1RcvFromC0_SlopeCaseLess2Deg_0 := 2258, txt_DbVar_C1_RamData4C1RcvFromC0_SlopeCaseLess4Deg_0 := 2259, txt_DbVar_C1_RamData4C1RcvFromC0_SlopeCaseLess6Deg_0 := 2260, txt_DbVar_C1_RamData4C1RcvFromC0_SlopeCaseHigher6Deg_0 := 2261, txt_DbVar_C1_RamData4C1RcvFromC0_TurretInSpeedZone2Deg_0 := 2262, txt_DbVar_C1_RamData4C1RcvFromC0_TurretInSpeedZone4Deg_0 := 2263, txt_DbVar_C1_RamData4C1RcvFromC0_TurretInSpeedZone2DegForBasket_0 := 2264, txt_DbVar_C1_RamData4C1RcvFromC0_SelectedControlPost_0 := 2265, txt_DbVar_C1_RamData4C1RcvFromC0_UpMastSensorNC_0 := 2266, txt_DbVar_C1_RamData4C1RcvFromC0_ValveInDownPositionSensor_0 := 2267, txt_DbVar_C1_RamData4C1RcvFromC0_MeasuringMastSensorFolded_0 := 2268, txt_DbVar_C1_RamData4C1RcvFromC0_PresenceSensorPlate_0 := 2269, txt_DbVar_C1_RamData4C1RcvFromC0_RecoveryReductionRatio_0 := 2270, txt_DbVar_C1_RamGeneralNeotecC1_RamGeneralNeotecC1_1_0 := 2271, txt_DbVar_C1_RamGeneralNeotecC1_RamGeneralNeotecC1_1_1_0 := 2272, txt_DbVar_C1_RamGeneralNeotecC1_RamGeneralNeotecC1_1_2_0 := 2273, txt_DbVar_C1_RamGeneralNeotecC1_RamGeneralNeotecC1_1_3_0 := 2274, txt_DbVar_C1_RamGeneralNeotecC1_RamGeneralNeotecC1_1_4_0 := 2275, txt_DbVar_C1_RamGeneralNeotecC1_RamGeneralNeotecC1_1_5_0 := 2276, txt_DbVar_C1_RamGeneralNeotecC1_RamGeneralNeotecC1_1_6_0 := 2277, txt_DbVar_C1_RamGeneralNeotecC1_RamGeneralNeotecC1_1_7_0 := 2278, txt_DbVar_C1_RamGeneralNeotecC1_RamGeneralNeotecC1_1_8_0 := 2279, txt_DbVar_C1_RamGeneralNeotecC1_RamGeneralNeotecC1_1_9_0 := 2280, txt_DbVar_C1_RamGeneralNeotecC1_RamGeneralNeotecC1_1_10_0 := 2281, txt_DbVar_C1_RamGeneralNeotecC1_RamGeneralNeotecC1_1_11_0 := 2282, txt_DbVar_C1_RamGeneralNeotecC1_RamGeneralNeotecC1_1_12_0 := 2283, txt_DbVar_C1_RamGeneralNeotecC1_RamGeneralNeotecC1_1_13_0 := 2284, txt_DbVar_C1_RamGeneralNeotecC1_RamGeneralNeotecC1_1_14_0 := 2285, txt_DbVar_C1_RamGeneralNeotecC1_RamGeneralNeotecC1_1_15_0 := 2286, txt_DbVar_C1_RamGeneralNeotecC1_RamGeneralNeotecC1_2_0 := 2287, txt_DbVar_C1_RamGeneralNeotecC1_RamGeneralNeotecC1_2_1_0 := 2288, txt_DbVar_C1_RamGeneralNeotecC1_RamGeneralNeotecC1_2_2_0 := 2289, txt_DbVar_C1_RamGeneralNeotecC1_RamGeneralNeotecC1_2_3_0 := 2290, txt_DbVar_C1_RamGeneralNeotecC1_RamGeneralNeotecC1_2_4_0 := 2291, txt_DbVar_C1_RamGeneralNeotecC1_RamGeneralNeotecC1_2_5_0 := 2292, txt_DbVar_C1_RamGeneralNeotecC1_RamGeneralNeotecC1_3_0 := 2293, txt_DbVar_C1_RamGeneralNeotecC1_RamGeneralNeotecC1_3_1_0 := 2294, txt_DbVar_C1_RamGeneralNeotecC1_RamGeneralNeotecC1_3_2_0 := 2295, txt_DbVar_C1_RamGeneralNeotecC1_RamGeneralNeotecC1_3_3_0 := 2296, txt_DbVar_C1_RamGeneralNeotecC1_RamGeneralNeotecC1_3_4_0 := 2297, txt_DbVar_C1_RamGeneralNeotecC1_RamGeneralNeotecC1_3_5_0 := 2298, txt_DbVar_C1_RamGeneralNeotecC1_RamGeneralNeotecC1_3_6_0 := 2299, txt_DbVar_C1_RamGeneralNeotecC1_RamGeneralNeotecC1_3_7_0 := 2300, txt_DbVar_C1_RamGeneralNeotecC1_RamGeneralNeotecC1_3_8_0 := 2301, txt_DbVar_C1_RamGeneralNeotecC1_RamGeneralNeotecC1_4_0 := 2302, txt_DbVar_C1_RamGeneralNeotecC1_RamGeneralNeotecC1_4_1_0 := 2303, txt_DbVar_C1_RamGeneralNeotecC1_RamGeneralNeotecC1_4_2_0 := 2304, txt_DbVar_C1_RamGeneralNeotecC1_RamGeneralNeotecC1_4_3_0 := 2305, txt_DbVar_C1_RamGeneralNeotecC1_RamGeneralNeotecC1_4_4_0 := 2306, txt_DbVar_C1_RamGeneralNeotecC1_RamGeneralNeotecC1_4_5_0 := 2307, txt_DbVar_C1_RamGeneralNeotecC1_RamGeneralNeotecC1_4_6_0 := 2308, txt_DbVar_C1_RamGeneralNeotecC1_RamGeneralNeotecC1_4_7_0 := 2309, txt_DbVar_C1_RamGeneralNeotecC1_RamGeneralNeotecC1_4_8_0 := 2310, txt_DbVar_C1_RamGeneralNeotecC1_WaterTempJ1939_0 := 2311, txt_DbVar_C1_RamGeneralNeotecC1_OilPressureJ1939_0 := 2312, txt_DbVar_C1_RamGeneralNeotecC1_MotorSpeedJ1939_0 := 2313, txt_DbVar_C1_RamGeneralNeotecC1_AlternatorCurentJ1939_0 := 2314, txt_DbVar_C1_RamGeneralNeotecC1_MotorStateJ1939_0 := 2315, txt_DbVar_C1_RamGeneralNeotecC1_PowerBatterie_0 := 2316, txt_DbVar_C1_RamGeneralNeotecC1_MotorSpeedCmdJ1939_0 := 2317, txt_DbVar_C1_RamGeneralNeotecC1_OverrideControlModeCmdJ1939_0 := 2318, txt_DbVar_C1_RamGeneralNeotecC1_HighPressureOilJ1939_0 := 2319, txt_DbVar_C1_RamGeneralNeotecC1_WarmingActiveJ1939_0 := 2320, txt_DbVar_C1_RamGeneralNeotecC1_StopMotorJ1939_0 := 2321, txt_DbVar_C1_NvParamGreenEffC1_REGEN_SOC_FULL_0 := 2322, txt_DbVar_C1_NvParamGreenEffC1_REGEN_SOC_MAX_0 := 2323, txt_DbVar_C1_NvParamGreenEffC1_REGEN_HYST_SOC_MAX_0 := 2324, txt_DbVar_C1_NvParamGreenEffC1_NBR_REGEN_SOC_ALARM_0 := 2325, txt_DbVar_C1_NvParamGreenEffC1_NBR_REGEN_SOC_OVERED_0 := 2326, txt_DbVar_C1_NvParamGreenEffC1_ELECTRIC_MOTOR_RPM_MAX_0 := 2327, txt_DbVar_C1_NvParamGreenEffC1_ELECTRIC_MOTOR_RPM_MIN_0 := 2328, txt_DbVar_C1_NvParamGreenEffC1_ELECTRIC_MOTOR_RPM_PVG_0 := 2329, txt_DbVar_C1_NvParamGreenEffC1_ELECTRIC_MOTOR_RPM_TOR_0 := 2330, txt_DbVar_C1_NvParamGreenEffC1_ELECTRIC_MOTOR_COLD_OIL_TEMP_0 := 2331, txt_DbVar_C1_NvParamGreenEffC1_BATTERY_CAPACITY_AMP_HOUR_0 := 2332, txt_DbVar_C1_NvParamGreenEffC1_NbElementRemainingRegenTime_0 := 2333, txt_DbVar_C1_RamGreenEffC1_AlarmCptNbrRegenFinish_0 := 2334, txt_DbVar_C1_RamGreenEffC1_ElectricMotorForbidden_0 := 2335, txt_DbVar_C1_RamGreenEffC1_ColdOilTankTemperature_0 := 2336, txt_DbVar_C1_RamGreenEffC1_RpmMvtsElectricMode_0 := 2337, txt_DbVar_C1_RamGreenEffC1_RpmTransRailElectricMode_0 := 2338, txt_DbVar_C1_RamGreenEffC1_RpmOilTankTemp_0 := 2339, txt_DbVar_C1_RamGreenEffC1_RpmMotorElectric_0 := 2340, txt_DbVar_C1_RamGreenEffC1_GeneratorOn_0 := 2341, txt_DbVar_C1_RamGreenEffC1_AutoModeActivate_0 := 2342, txt_DbVar_C1_RamGreenEffC1_SilenceModeActivate_0 := 2343, txt_DbVar_C1_RamGreenEffC1_ForcingModeActivate_0 := 2344, txt_DbVar_C1_RamGreenEffC1_ForcingRegenlow_0 := 2345, txt_DbVar_C1_RamGreenEffC1_ForcingRegenHigh_0 := 2346, txt_DbVar_C1_RamGreenEffC1_RemainingRegenTimeAverage_0 := 2347, txt_DbVar_C1_RamGreenEffC1_AskReloadWithGenerator_0 := 2348, txt_DbVar_C1_RamGreenEffC1_ReloadWithGeneratorOn_0 := 2349, txt_DbVar_C1_RamGreenEffC1_SocStopRegen_0 := 2350, txt_DbVar_C1_RamGreenEffC1_TotalRegenHours_0 := 2351, txt_DbVar_C1_RamGreenEffC1_PictoColdOilTankTemperature_0 := 2352, txt_DbVar_C1_RamGreenEffC1_TotalElectricHours_0 := 2353, txt_DbVar_C1_RamGreenEffC1_PictoRecoveryReductionRatio_0 := 2354, txt_DbVarGrpName_FC_NV_PARAMERTERS_C0 := 2355, txt_DbVarGrpName_FC_NV_PARAM_SPEED_MAX_RAIL := 2356, txt_DbVarGrpName_FC_NV_PARAM_BRAKE_TEST := 2357, txt_DbVarGrpName_FC_NV_PARAM_RAIL_WORK_SAFETY_C0 := 2358, txt_DbVarGrpName_FC_NV_PARAM_TRANSPORT_POS_C0 := 2359, txt_DbVarGrpName_FC_NV_PARAM_SELECT_CONTROL_POST := 2360, txt_DbVarGrpName_FC_NV_PARAM_ALARM_C0 := 2361, txt_DbVarGrpName_FC_NV_PARAM_MAST_DISPLAY_C0 := 2362, txt_DbVarGrpName_FC_NV_PARAMERTERS_C1 := 2363, txt_DbVarGrpName_FC_NV_PARAM_MOTOR_C1 := 2364, txt_DbVarGrpName_FC_NV_PARAM_LIMIT_WORK_ENVLP_C1 := 2365, txt_DbVarGrpName_FC_NV_PARAM_MVT_END_STOP_C1 := 2366, txt_DbVarGrpName_FC_NV_PARAM_AUTO_STOP_C1 := 2367, txt_DbVarGrpName_FC_NV_PARAM_MAST_C1 := 2368, txt_DbVarGrpName_FC_NV_PARAM_ALARM_C1 := 2369, txt_DbVarGrpName_FC_NV_OPTION_C0 := 2370, txt_DbVarGrpName_FC_NV_OPTION_C1 := 2371) UINT;
END_TYPE

